TYPE ServicesTimingIOStatuses :
STRUCT
	///Is the I/O in a healthy state?
	healthStatus: HealthStatus;
END_STRUCT
END_TYPE

(* stored: Version 1.1.0.1, ProductVersion 3.1.4019.2
   DUT ServicesTimingIOStatuses: Id {23c66b63-dee7-4049-8d85-4a8039367570} *)
